Omron CX-Programmer project NewProject (CX-Programmer 9.75)

# PLC Memory: CP1E N30

## Program NewProgram1 (cyclic task 0)
Local symbols
M0 10.00 BOOL  ; 10.00
M1 10.01 BOOL  ; 10.01
M2 10.02 BOOL  ; 10.02
M3 10.03 BOOL  ; 10.03
Output 100.00 BOOL  ; 100.00
PB 0.00 BOOL  ; 0.00
PB1 0.01 BOOL  ; 0.01

### Section Section1

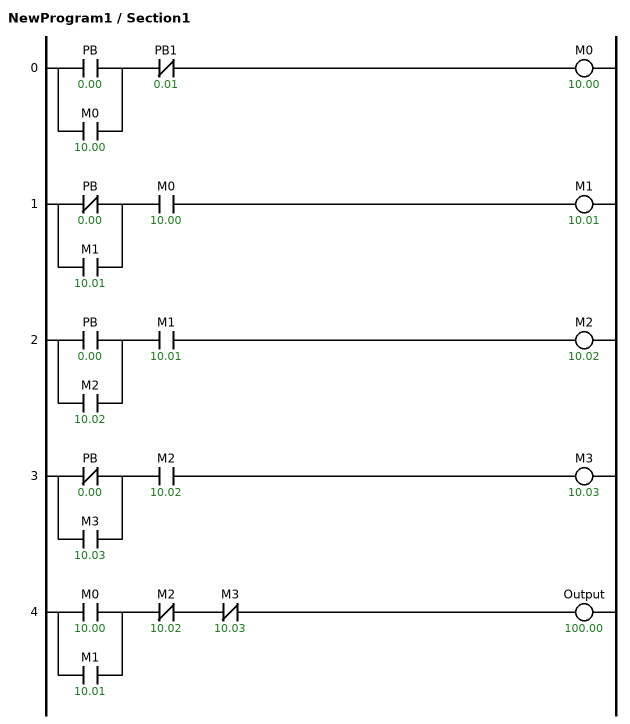
; rung 0
LD PB  ; 0.00
OR M0  ; 10.00
ANDNOT PB1  ; 0.01
OUT M0  ; 10.00
; rung 1
LDNOT PB  ; 0.00
OR M1  ; 10.01
AND M0  ; 10.00
OUT M1  ; 10.01
; rung 2
LD PB  ; 0.00
OR M2  ; 10.02
AND M1  ; 10.01
OUT M2  ; 10.02
; rung 3
LDNOT PB  ; 0.00
OR M3  ; 10.03
AND M2  ; 10.02
OUT M3  ; 10.03
; rung 4
LD M0  ; 10.00
OR M1  ; 10.01
ANDNOT M2  ; 10.02
ANDNOT M3  ; 10.03
OUT Output  ; 100.00

### Section END
; rung 0
END(001)